(* Logix 5000 project; controller SX_V040001_C001 vendor 1 type 14 code 77 rev 16.23; software revision 16.04; part 13 of 35 *)
(* tags used below, declared in another part *)
   ALL_KINDS : INT[90];
   DB_A_IO : INT[16];
   DB_D_IO : DINT[6];
   DB_D_IO_REVERSE : DINT[6];
   DRIVE : INT[32];
   EMPTYING : INT[18];
   G_AInput : DINT[8];
   G_DInput : DINT[3];
   G_DOutput : DINT[3];
   loading : INT[19];
   louvre : INT[11];
   m_on_off_line : BOOL;
   METERING : INT[44];
   PARAMETER : INT[501];
   RM_CMD : INT[9];
   STATUS_GENERAL : INT[135];
   STATUS_SEND_PART_1 : INT[135];
   TEMP : INT[14];
(* MainProgram, continued *)

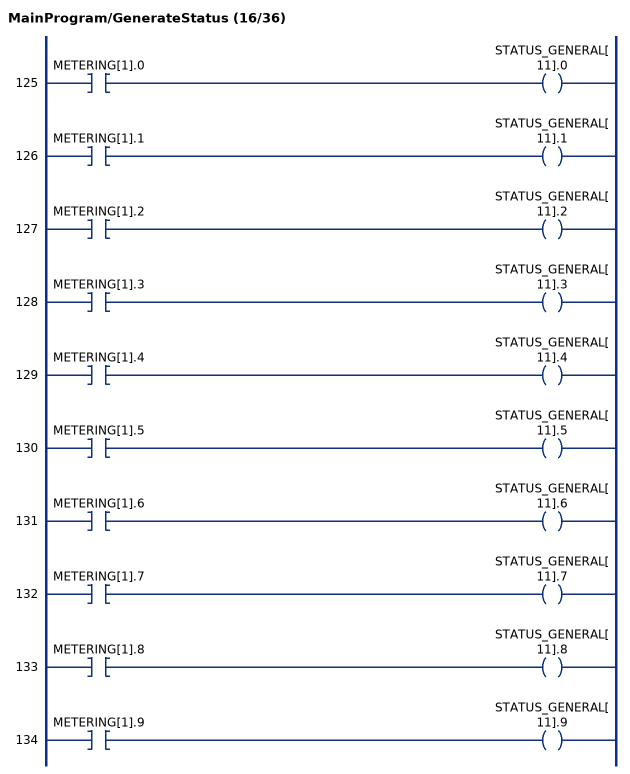
   [picture p280: MainProgram/GenerateStatus rungs 125-134]
   125: XIC(METERING[1].0)OTE(STATUS_GENERAL[11].0);
   126: XIC(METERING[1].1)OTE(STATUS_GENERAL[11].1);
   127: XIC(METERING[1].2)OTE(STATUS_GENERAL[11].2);
   128: XIC(METERING[1].3)OTE(STATUS_GENERAL[11].3);
   129: XIC(METERING[1].4)OTE(STATUS_GENERAL[11].4);
   130: XIC(METERING[1].5)OTE(STATUS_GENERAL[11].5);
   131: XIC(METERING[1].6)OTE(STATUS_GENERAL[11].6);
   132: XIC(METERING[1].7)OTE(STATUS_GENERAL[11].7);
   133: XIC(METERING[1].8)OTE(STATUS_GENERAL[11].8);
   134: XIC(METERING[1].9)OTE(STATUS_GENERAL[11].9);
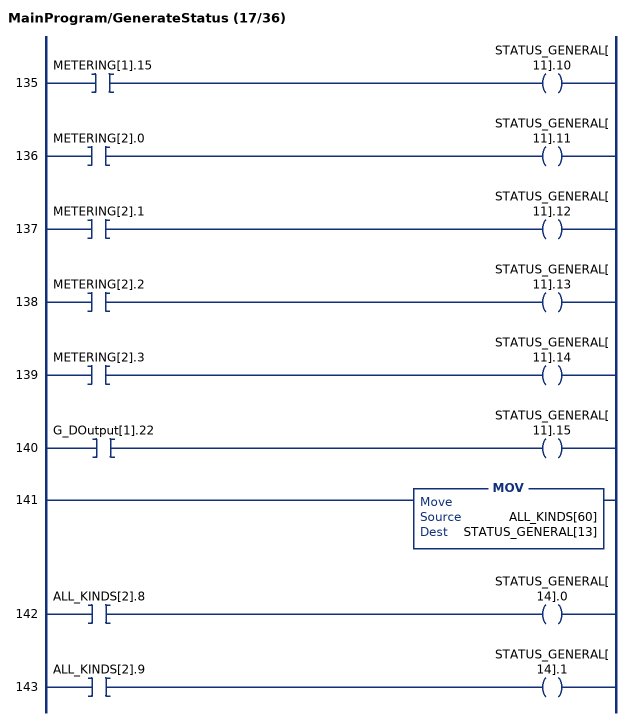
   135: XIC(METERING[1].15)OTE(STATUS_GENERAL[11].10);
   136: XIC(METERING[2].0)OTE(STATUS_GENERAL[11].11);
   137: XIC(METERING[2].1)OTE(STATUS_GENERAL[11].12);
   138: XIC(METERING[2].2)OTE(STATUS_GENERAL[11].13);
   139: XIC(METERING[2].3)OTE(STATUS_GENERAL[11].14);
   140: XIC(G_DOutput[1].22)OTE(STATUS_GENERAL[11].15);
   141: MOV(ALL_KINDS[60],STATUS_GENERAL[13]);
   142: XIC(ALL_KINDS[2].8)OTE(STATUS_GENERAL[14].0);
   143: XIC(ALL_KINDS[2].9)OTE(STATUS_GENERAL[14].1);
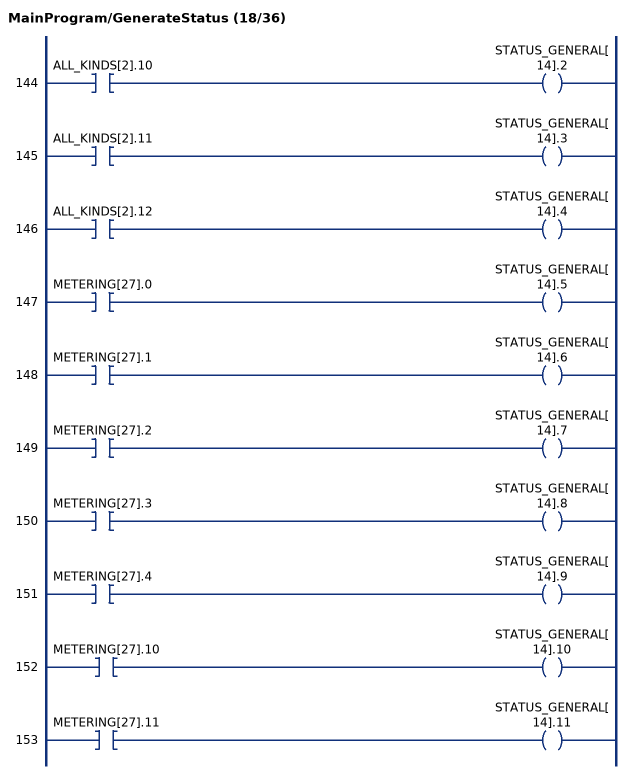
   144: XIC(ALL_KINDS[2].10)OTE(STATUS_GENERAL[14].2);
   145: XIC(ALL_KINDS[2].11)OTE(STATUS_GENERAL[14].3);
   146: XIC(ALL_KINDS[2].12)OTE(STATUS_GENERAL[14].4);
   147: XIC(METERING[27].0)OTE(STATUS_GENERAL[14].5);
   148: XIC(METERING[27].1)OTE(STATUS_GENERAL[14].6);
   149: XIC(METERING[27].2)OTE(STATUS_GENERAL[14].7);
   150: XIC(METERING[27].3)OTE(STATUS_GENERAL[14].8);
   151: XIC(METERING[27].4)OTE(STATUS_GENERAL[14].9);
   152: XIC(METERING[27].10)OTE(STATUS_GENERAL[14].10);
   153: XIC(METERING[27].11)OTE(STATUS_GENERAL[14].11);
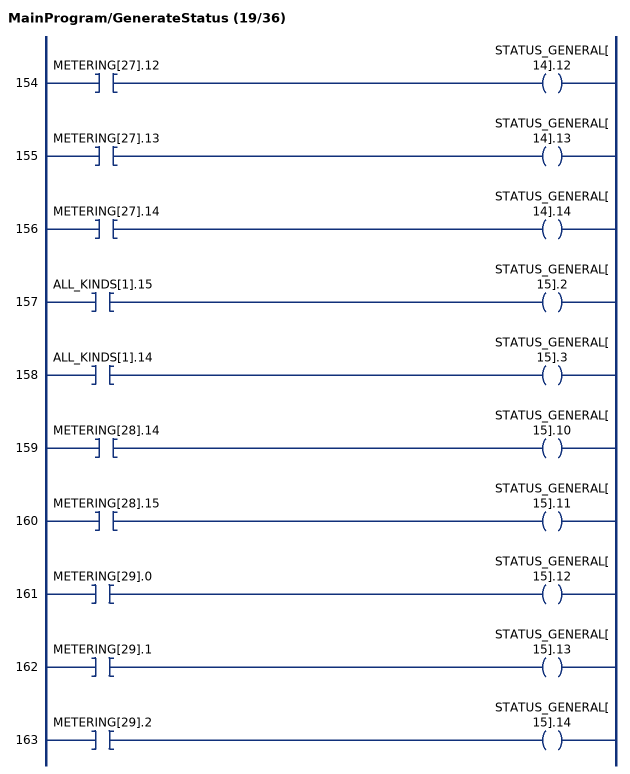
   154: XIC(METERING[27].12)OTE(STATUS_GENERAL[14].12);
   155: XIC(METERING[27].13)OTE(STATUS_GENERAL[14].13);
   156: XIC(METERING[27].14)OTE(STATUS_GENERAL[14].14);
   157: XIC(ALL_KINDS[1].15)OTE(STATUS_GENERAL[15].2);
   158: XIC(ALL_KINDS[1].14)OTE(STATUS_GENERAL[15].3);
   159: XIC(METERING[28].14)OTE(STATUS_GENERAL[15].10);
   160: XIC(METERING[28].15)OTE(STATUS_GENERAL[15].11);
   161: XIC(METERING[29].0)OTE(STATUS_GENERAL[15].12);
   162: XIC(METERING[29].1)OTE(STATUS_GENERAL[15].13);
   163: XIC(METERING[29].2)OTE(STATUS_GENERAL[15].14);
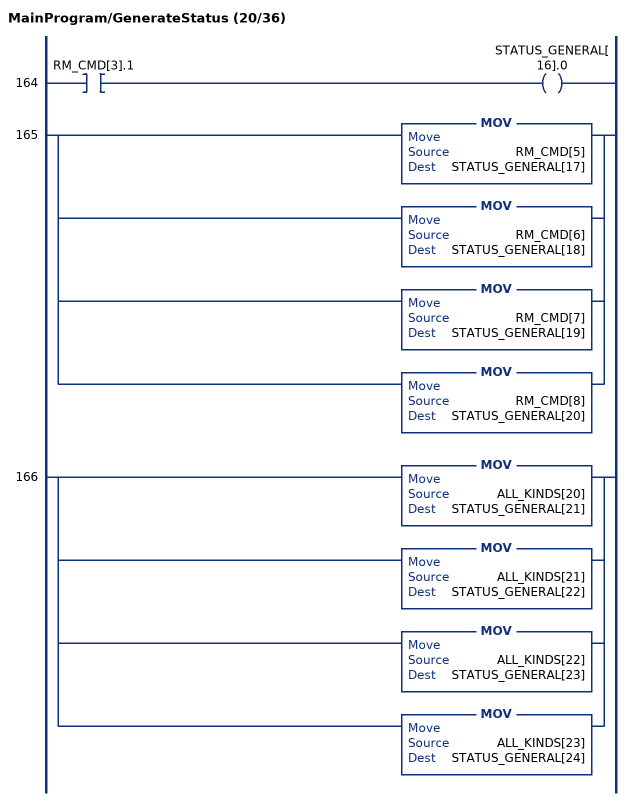
   164: XIC(RM_CMD[3].1)OTE(STATUS_GENERAL[16].0);
   165: [MOV(RM_CMD[5],STATUS_GENERAL[17]) ,MOV(RM_CMD[6],STATUS_GENERAL[18]) ,MOV(RM_CMD[7],STATUS_GENERAL[19]) ,MOV(RM_CMD[8],STATUS_GENERAL[20]) ];
   166: [MOV(ALL_KINDS[20],STATUS_GENERAL[21]) ,MOV(ALL_KINDS[21],STATUS_GENERAL[22]) ,MOV(ALL_KINDS[22],STATUS_GENERAL[23]) ,MOV(ALL_KINDS[23],STATUS_GENERAL[24]) ];
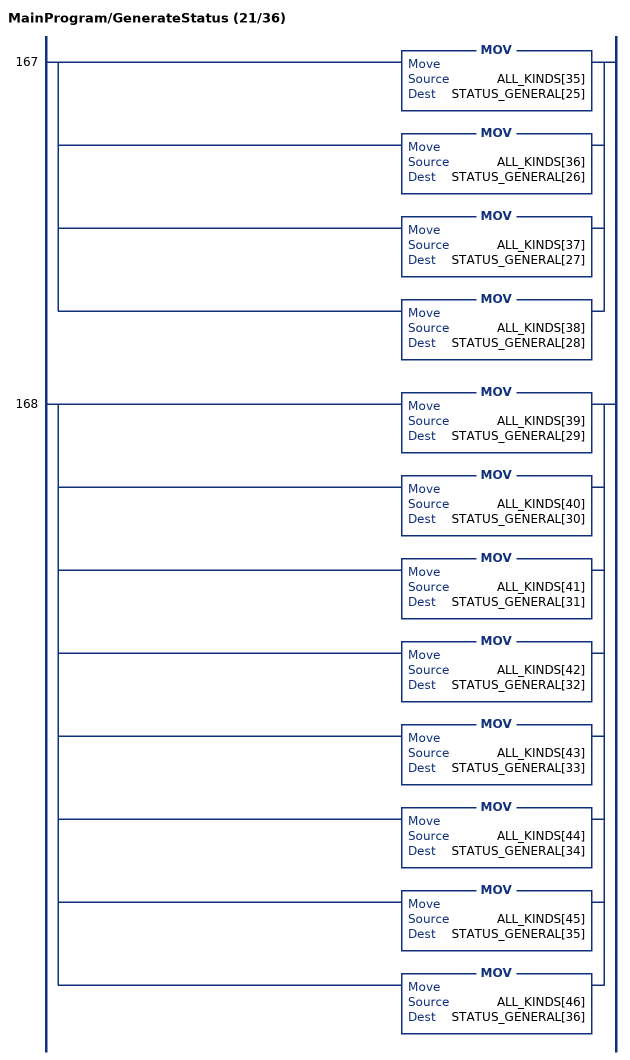
   167: [MOV(ALL_KINDS[35],STATUS_GENERAL[25]) ,MOV(ALL_KINDS[36],STATUS_GENERAL[26]) ,MOV(ALL_KINDS[37],STATUS_GENERAL[27]) ,MOV(ALL_KINDS[38],STATUS_GENERAL[28]) ];
   168: [MOV(ALL_KINDS[39],STATUS_GENERAL[29]) ,MOV(ALL_KINDS[40],STATUS_GENERAL[30]) ,MOV(ALL_KINDS[41],STATUS_GENERAL[31]) ,MOV(ALL_KINDS[42],STATUS_GENERAL[32]) ,MOV(ALL_KINDS[43],STATUS_GENERAL[33]) ,MOV(ALL_KINDS[44],STATUS_GENERAL[34]) ,MOV(ALL_KINDS[45],STATUS_GENERAL[35]) ,MOV(ALL_KINDS[46],STATUS_GENERAL[36]) ];
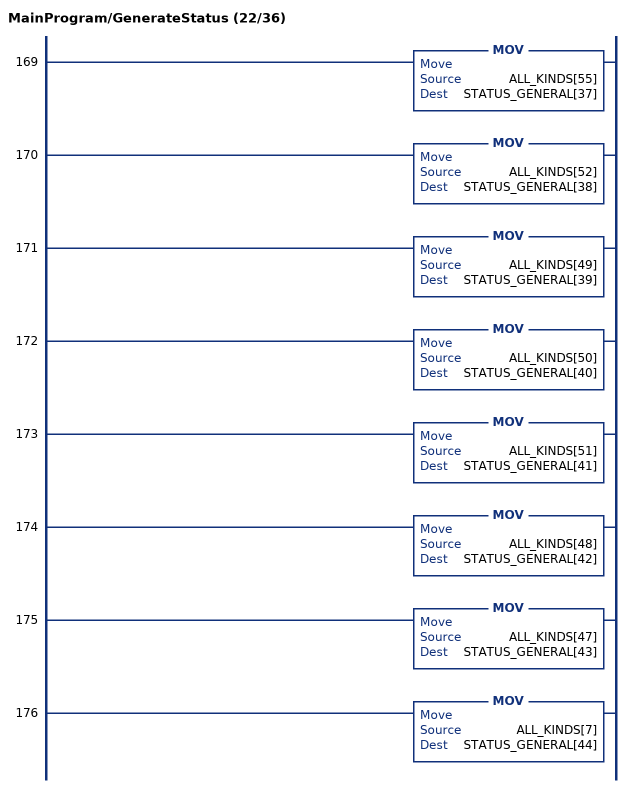
   169: MOV(ALL_KINDS[55],STATUS_GENERAL[37]);
   170: MOV(ALL_KINDS[52],STATUS_GENERAL[38]);
   171: MOV(ALL_KINDS[49],STATUS_GENERAL[39]);
   172: MOV(ALL_KINDS[50],STATUS_GENERAL[40]);
   173: MOV(ALL_KINDS[51],STATUS_GENERAL[41]);
   174: MOV(ALL_KINDS[48],STATUS_GENERAL[42]);
   175: MOV(ALL_KINDS[47],STATUS_GENERAL[43]);
   176: MOV(ALL_KINDS[7],STATUS_GENERAL[44]);
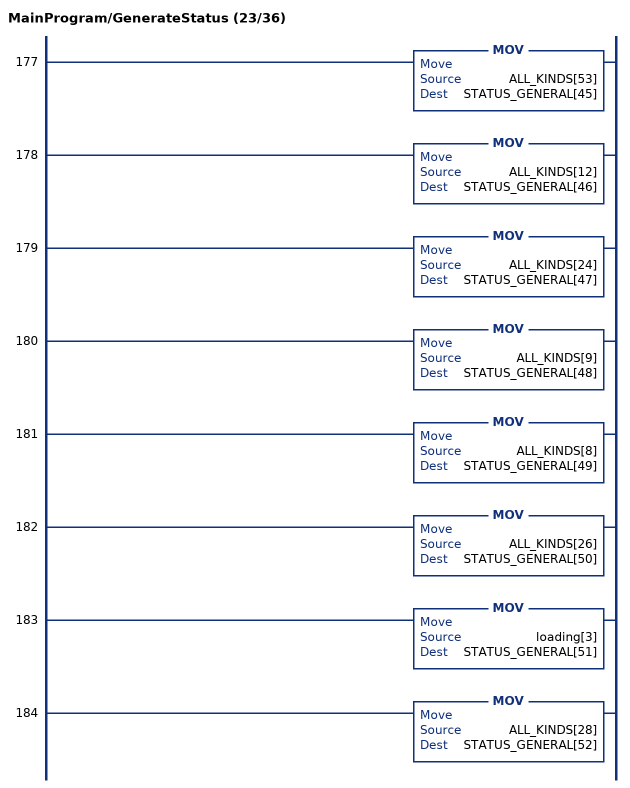
   177: MOV(ALL_KINDS[53],STATUS_GENERAL[45]);
   178: MOV(ALL_KINDS[12],STATUS_GENERAL[46]);
   179: MOV(ALL_KINDS[24],STATUS_GENERAL[47]);
   180: MOV(ALL_KINDS[9],STATUS_GENERAL[48]);
   181: MOV(ALL_KINDS[8],STATUS_GENERAL[49]);
   182: MOV(ALL_KINDS[26],STATUS_GENERAL[50]);
   183: MOV(loading[3],STATUS_GENERAL[51]);
   184: MOV(ALL_KINDS[28],STATUS_GENERAL[52]);
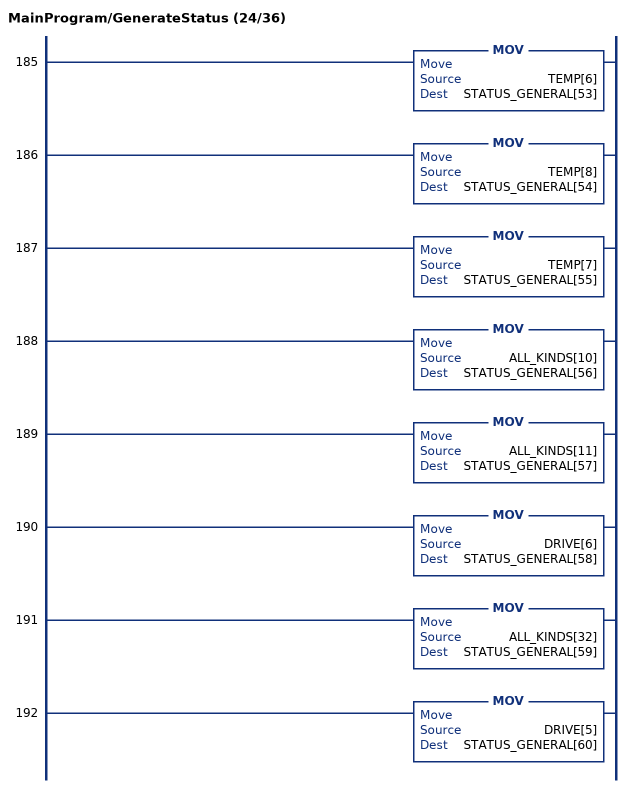
   185: MOV(TEMP[6],STATUS_GENERAL[53]);
   186: MOV(TEMP[8],STATUS_GENERAL[54]);
   187: MOV(TEMP[7],STATUS_GENERAL[55]);
   188: MOV(ALL_KINDS[10],STATUS_GENERAL[56]);
   189: MOV(ALL_KINDS[11],STATUS_GENERAL[57]);
   190: MOV(DRIVE[6],STATUS_GENERAL[58]);
   191: MOV(ALL_KINDS[32],STATUS_GENERAL[59]);
   192: MOV(DRIVE[5],STATUS_GENERAL[60]);
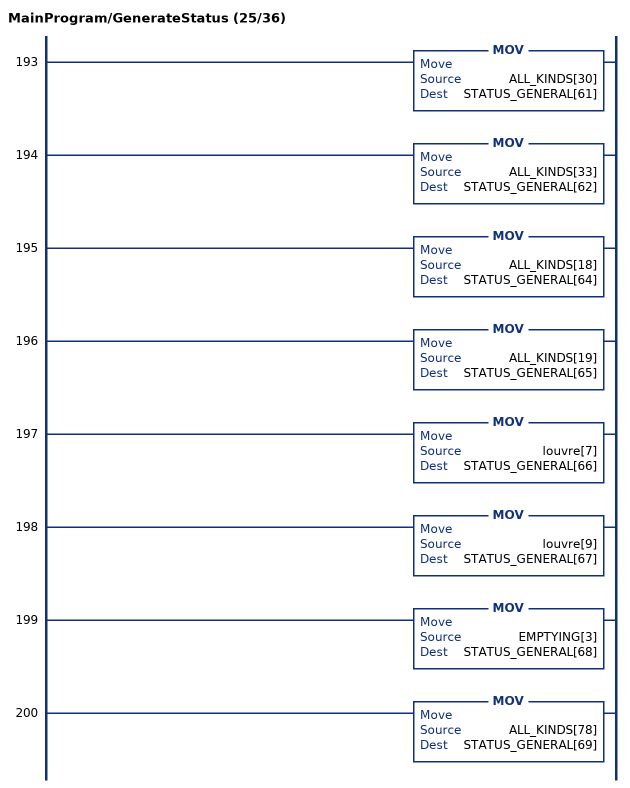
   193: MOV(ALL_KINDS[30],STATUS_GENERAL[61]);
   194: MOV(ALL_KINDS[33],STATUS_GENERAL[62]);
   195: MOV(ALL_KINDS[18],STATUS_GENERAL[64]);
   196: MOV(ALL_KINDS[19],STATUS_GENERAL[65]);
   197: MOV(louvre[7],STATUS_GENERAL[66]);
   198: MOV(louvre[9],STATUS_GENERAL[67]);
   199: MOV(EMPTYING[3],STATUS_GENERAL[68]);
   200: MOV(ALL_KINDS[78],STATUS_GENERAL[69]);
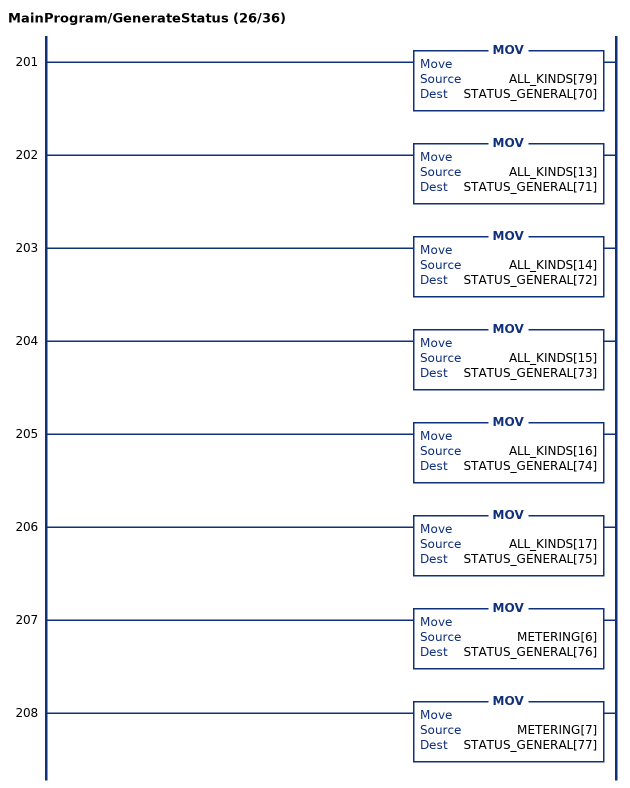
   201: MOV(ALL_KINDS[79],STATUS_GENERAL[70]);
   202: MOV(ALL_KINDS[13],STATUS_GENERAL[71]);
   203: MOV(ALL_KINDS[14],STATUS_GENERAL[72]);
   204: MOV(ALL_KINDS[15],STATUS_GENERAL[73]);
   205: MOV(ALL_KINDS[16],STATUS_GENERAL[74]);
   206: MOV(ALL_KINDS[17],STATUS_GENERAL[75]);
   207: MOV(METERING[6],STATUS_GENERAL[76]);
   208: MOV(METERING[7],STATUS_GENERAL[77]);
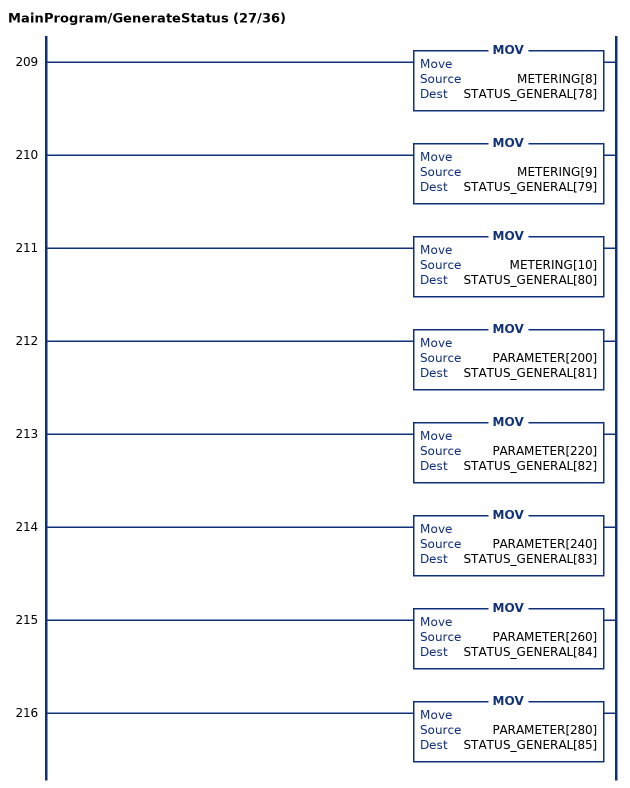
   209: MOV(METERING[8],STATUS_GENERAL[78]);
   210: MOV(METERING[9],STATUS_GENERAL[79]);
   211: MOV(METERING[10],STATUS_GENERAL[80]);
   212: MOV(PARAMETER[200],STATUS_GENERAL[81]);
   213: MOV(PARAMETER[220],STATUS_GENERAL[82]);
   214: MOV(PARAMETER[240],STATUS_GENERAL[83]);
   215: MOV(PARAMETER[260],STATUS_GENERAL[84]);
   216: MOV(PARAMETER[280],STATUS_GENERAL[85]);
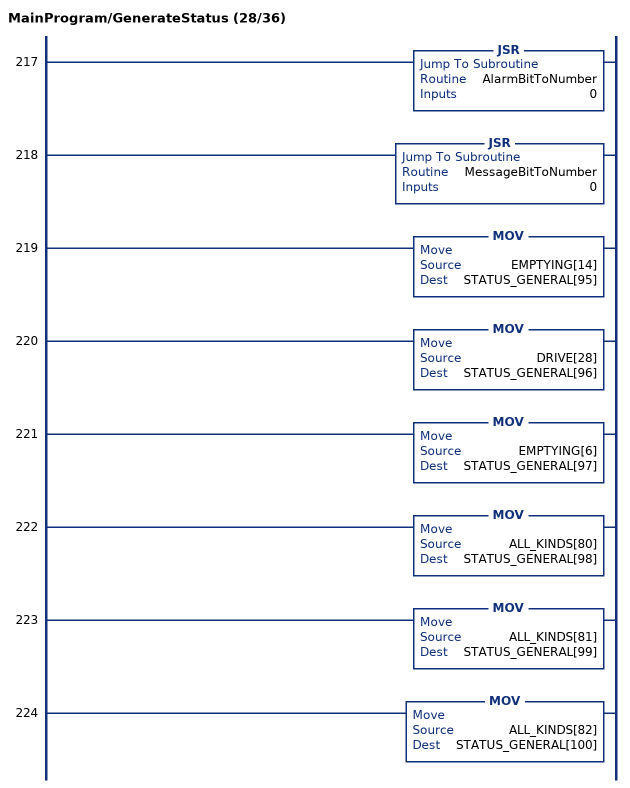
   217: JSR(AlarmBitToNumber,0);
   218: JSR(MessageBitToNumber,0);
   219: MOV(EMPTYING[14],STATUS_GENERAL[95]);
   220: MOV(DRIVE[28],STATUS_GENERAL[96]);
   221: MOV(EMPTYING[6],STATUS_GENERAL[97]);
   222: MOV(ALL_KINDS[80],STATUS_GENERAL[98]);
   223: MOV(ALL_KINDS[81],STATUS_GENERAL[99]);
   224: MOV(ALL_KINDS[82],STATUS_GENERAL[100]);
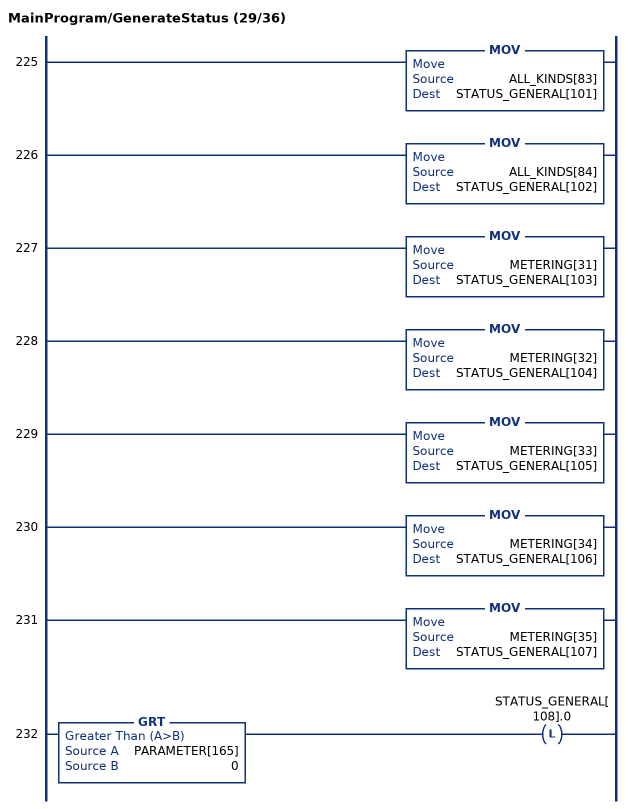
   225: MOV(ALL_KINDS[83],STATUS_GENERAL[101]);
   226: MOV(ALL_KINDS[84],STATUS_GENERAL[102]);
   227: MOV(METERING[31],STATUS_GENERAL[103]);
   228: MOV(METERING[32],STATUS_GENERAL[104]);
   229: MOV(METERING[33],STATUS_GENERAL[105]);
   230: MOV(METERING[34],STATUS_GENERAL[106]);
   231: MOV(METERING[35],STATUS_GENERAL[107]);
   232: GRT(PARAMETER[165],0)OTL(STATUS_GENERAL[108].0);
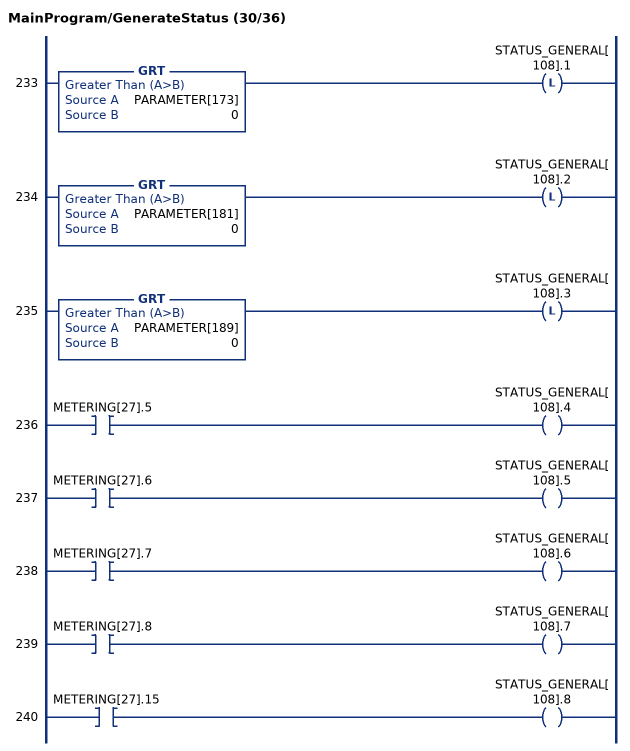
   233: GRT(PARAMETER[173],0)OTL(STATUS_GENERAL[108].1);
   234: GRT(PARAMETER[181],0)OTL(STATUS_GENERAL[108].2);
   235: GRT(PARAMETER[189],0)OTL(STATUS_GENERAL[108].3);
   236: XIC(METERING[27].5)OTE(STATUS_GENERAL[108].4);
   237: XIC(METERING[27].6)OTE(STATUS_GENERAL[108].5);
   238: XIC(METERING[27].7)OTE(STATUS_GENERAL[108].6);
   239: XIC(METERING[27].8)OTE(STATUS_GENERAL[108].7);
   240: XIC(METERING[27].15)OTE(STATUS_GENERAL[108].8);
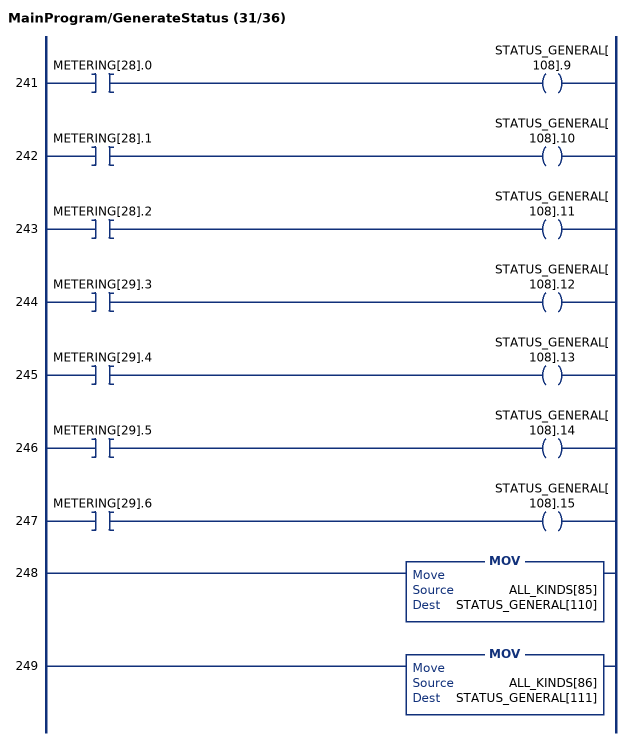
   241: XIC(METERING[28].0)OTE(STATUS_GENERAL[108].9);
   242: XIC(METERING[28].1)OTE(STATUS_GENERAL[108].10);
   243: XIC(METERING[28].2)OTE(STATUS_GENERAL[108].11);
   244: XIC(METERING[29].3)OTE(STATUS_GENERAL[108].12);
   245: XIC(METERING[29].4)OTE(STATUS_GENERAL[108].13);
   246: XIC(METERING[29].5)OTE(STATUS_GENERAL[108].14);
   247: XIC(METERING[29].6)OTE(STATUS_GENERAL[108].15);
   248: MOV(ALL_KINDS[85],STATUS_GENERAL[110]);
   249: MOV(ALL_KINDS[86],STATUS_GENERAL[111]);
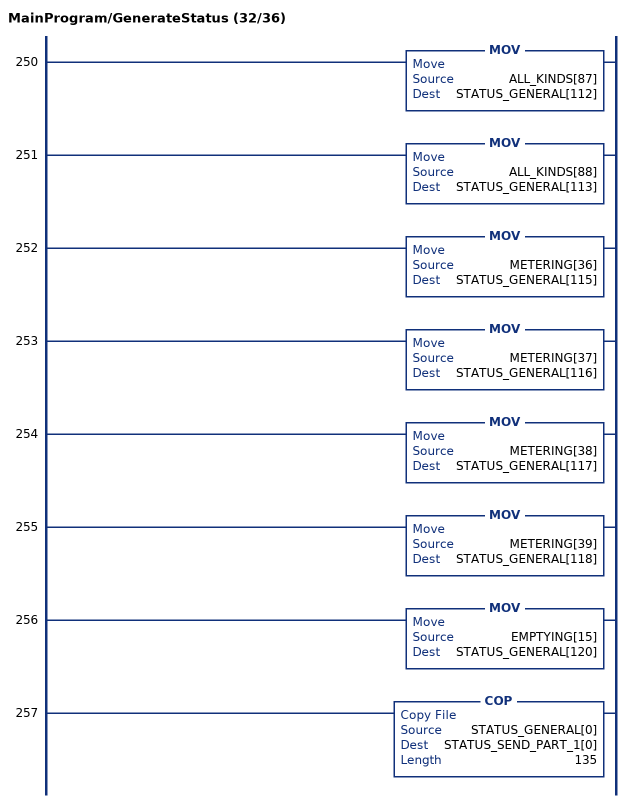
   250: MOV(ALL_KINDS[87],STATUS_GENERAL[112]);
   251: MOV(ALL_KINDS[88],STATUS_GENERAL[113]);
   252: MOV(METERING[36],STATUS_GENERAL[115]);
   253: MOV(METERING[37],STATUS_GENERAL[116]);
   254: MOV(METERING[38],STATUS_GENERAL[117]);
   255: MOV(METERING[39],STATUS_GENERAL[118]);
   256: MOV(EMPTYING[15],STATUS_GENERAL[120]);
   257: COP(STATUS_GENERAL[0],STATUS_SEND_PART_1[0],135);
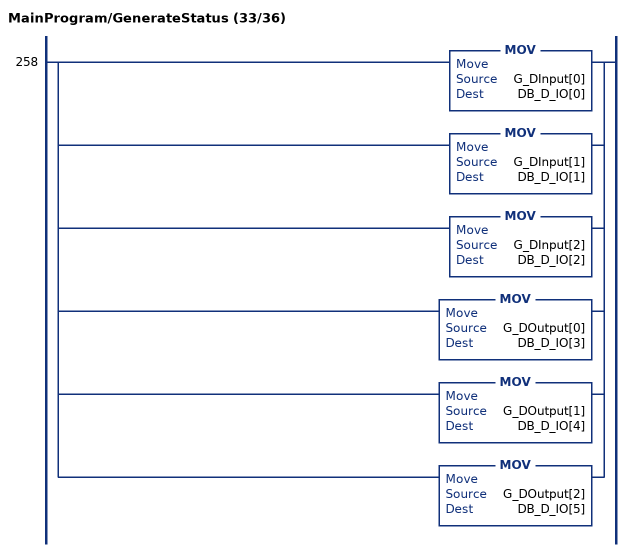
   258: [MOV(G_DInput[0],DB_D_IO[0]) ,MOV(G_DInput[1],DB_D_IO[1]) ,MOV(G_DInput[2],DB_D_IO[2]) ,MOV(G_DOutput[0],DB_D_IO[3]) ,MOV(G_DOutput[1],DB_D_IO[4]) ,MOV(G_DOutput[2],DB_D_IO[5]) ];
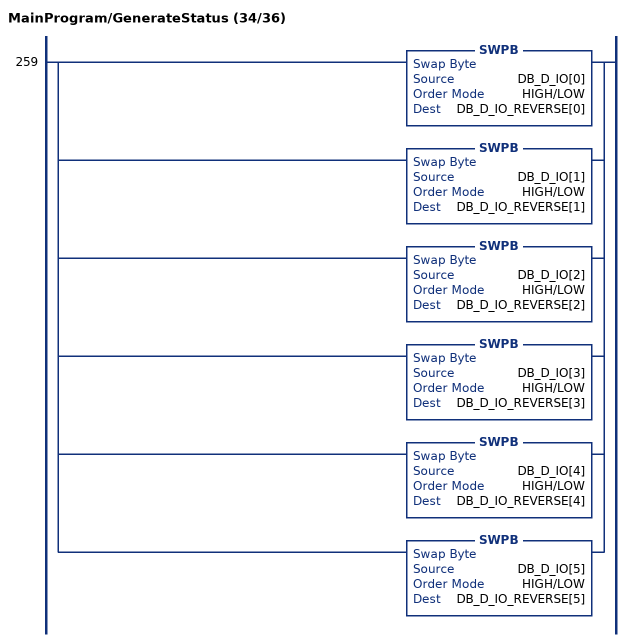
   259: [SWPB(DB_D_IO[0],HIGH/LOW,DB_D_IO_REVERSE[0]) ,SWPB(DB_D_IO[1],HIGH/LOW,DB_D_IO_REVERSE[1]) ,SWPB(DB_D_IO[2],HIGH/LOW,DB_D_IO_REVERSE[2]) ,SWPB(DB_D_IO[3],HIGH/LOW,DB_D_IO_REVERSE[3]) ,SWPB(DB_D_IO[4],HIGH/LOW,DB_D_IO_REVERSE[4]) ,SWPB(DB_D_IO[5],HIGH/LOW,DB_D_IO_REVERSE[5]) ];
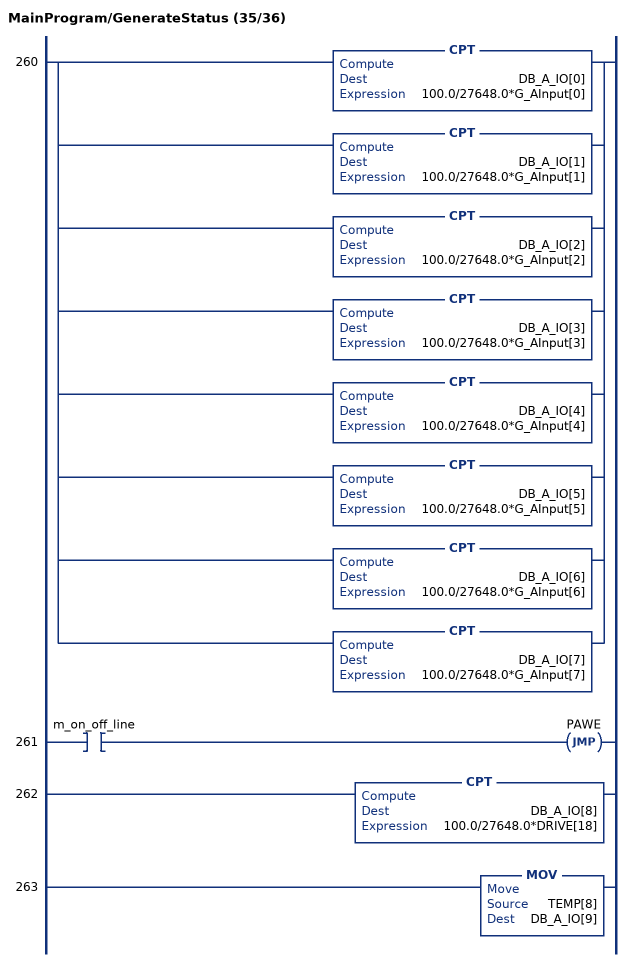
   260: [CPT(DB_A_IO[0],100.0/27648.0*G_AInput[0]) ,CPT(DB_A_IO[1],100.0/27648.0*G_AInput[1]) ,CPT(DB_A_IO[2],100.0/27648.0*G_AInput[2]) ,CPT(DB_A_IO[3],100.0/27648.0*G_AInput[3]) ,CPT(DB_A_IO[4],100.0/27648.0*G_AInput[4]) ,CPT(DB_A_IO[5],100.0/27648.0*G_AInput[5]) ,CPT(DB_A_IO[6],100.0/27648.0*G_AInput[6]) ,CPT(DB_A_IO[7],100.0/27648.0*G_AInput[7]) ];
   261: XIC(m_on_off_line)JMP(PAWE);
   262: CPT(DB_A_IO[8],100.0/27648.0*DRIVE[18]);
   263: MOV(TEMP[8],DB_A_IO[9]);
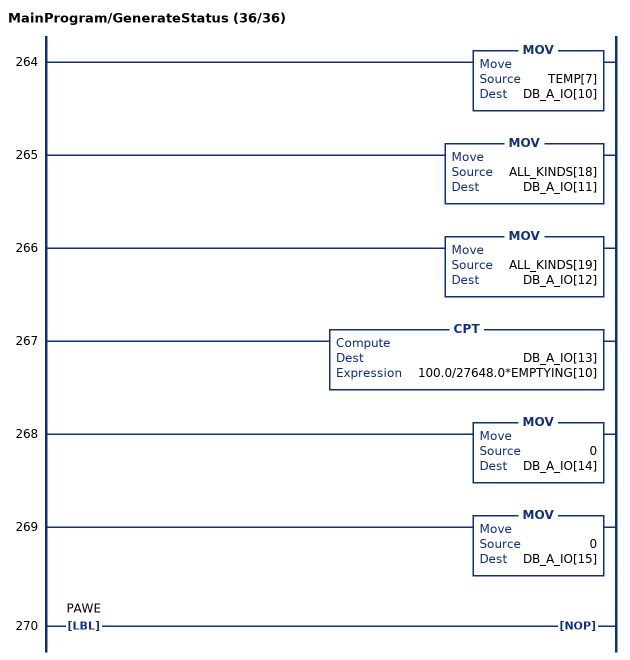
   264: MOV(TEMP[7],DB_A_IO[10]);
   265: MOV(ALL_KINDS[18],DB_A_IO[11]);
   266: MOV(ALL_KINDS[19],DB_A_IO[12]);
   267: CPT(DB_A_IO[13],100.0/27648.0*EMPTYING[10]);
   268: MOV(0,DB_A_IO[14]);
   269: MOV(0,DB_A_IO[15]);
   270: LBL(PAWE)NOP();
END_ROUTINE
